# B&R Automation Studio project mappLogbook
Automation Studio 4.7.5.60 SP; technology packages: mappView 5.11.3

## Configuration PC

CPU X20CP1583, AutomationRuntime C4.72, Build 4.1.2, Safety 0.0, Vc V4.52.0

### Task classes (Cpu.sw)
```
Cyclic#8:
  Logbook <- mappLogbook.Logbook.prg
Binaries: mvLoader, TCData, udbdef, User, asfw, OpcUaMap, iomap, sysconf, arconfig, ashwd, Role, ashwac
Libraries: runtime, AsBrStr, asieccon, fileio, IecCheck, sys_lib, ArEventLog, astime
```

### Hardware
```
X20CP1583 : X20CP1583 v1.6.0.0
  Connector IF1:
    ActivateIna = 0
  Connector IF2:
    ActivateDevice = 1
  ConfigurationID = ARuser_PC
  Simulation = 1
  VolatileGlobalPvSize = 200000
  Cyclic3Tolerance = 60000000
  FileDevice1
  FileDeviceName1 = FileDevice
  FileDevicePath1 = C:\Users\hendricksf\Desktop
  ActivateOpcUa = 1
  OpcUaInformationModels_PV_Version = 1
```

## Logical view

Binary libraries used (declarations not repeated): operator, runtime, AsIecCon, AsBrStr, IecCheck, sys_lib, ArEventLog, astime, AsHttp, standard

### Package Logical/Libraries - Globale Bibliotheken

- Visualisation Logical/mappView (not shown)

### LogTypes.typ
```iecst
TYPE
	enumLogbookState :
		( (*State machine*)
		stateWait,
		stateOpen,
		stateLatest,
		stateNext,
		stateDetails1,
		stateDetails2,
		stateDetails3,
		stateDetails4,
		stateFilter,
		statePrep,
		stateError,
		stateNone
		);
	enumSeverity :
		(
		severityNotification,
		severityInformation,
		severityWarning,
		severityError
		);
	enumLogbookType :
		(
		logAccessSecurity,
		logCommisioning,
		logConnectivity,
		logFieldbus,
		logFirewall,
		logMapp,
		logMotion,
		logSafety,
		logSystem,
		logTextSystem,
		logUnitSystem,
		logUser,
		logVisualization
		);
	enumSorting :
		(
		sortingASC,
		sortingDESC
		);
	logbookCMD : 	STRUCT  (*Command structure*)
		Refresh : BOOL; (*Read all entries*)
		Update : BOOL; (*Update entries*)
		Write : BOOL; (*Write a new entry*)
		ResetError : BOOL; (*Reset error*)
	END_STRUCT;
	logbookPAR : 	STRUCT  (*Parameter structure*)
		DateNow : DATE_AND_TIME; (*Current date and time*)
		TableConfig : STRING[100]; (*Hide unused rows*)
		EntriesMax : UINT; (*Maximum number of entries, shadow of LOGBOOK_ENTRIES_MAX*)
		FilterErrorNo : UDINT; (*Filter by error number*)
		FilterErrorText : STRING[LOGBOOK_TEXT_LEN]; (*Filter by error text*)
		FilterSeverity : ARRAY[0..3]OF BOOL := [4(TRUE)]; (*Filter by severity*)
		FilterLogbook : ARRAY[0..LOGBOOK_BOOKS_MAX]OF BOOL := [14(TRUE)]; (*Filter by logbook*)
		FilterDateStart : DATE; (*Filter by date*)
		FilterDateEnd : DATE;
		Sorting : enumSorting := sortingDESC; (*Sort date asc or desc*)
		AbortOnEntriesLimit : BOOL; (*Stop looking for additional entries when limit is reached*)
		AutoUpdate : BOOL; (*Automatically update data*)
		AutoUpdateInterval : UINT := 60; (*Interval for auto update in s*)
		WriteErrorNo : UDINT; (*Error no for new entry*)
		WriteErrorText : STRING[LOGBOOK_TEXT_LEN]; (*Error text for new entry*)
		WriteSeverity : USINT := 0; (*Error severiry for new entry*)
		WriteLogbook : UINT := 0; (*Error logbook for new entry*)
	END_STRUCT;
	logbookERR : 	STRUCT  (*Error structure*)
		State : enumLogbookState; (*State where the error occured*)
	END_STRUCT;
	logbookDAT : 	STRUCT  (*Data structure*)
		Entries : logbookENTRIES;
		EntriesTotal : UINT; (*Total number of entries*)
		CntSeverity : ARRAY[0..3]OF UINT; (*Counts by severity*)
		CntLogbook : ARRAY[0..LOGBOOK_BOOKS_MAX]OF UINT; (*Counts by logbook*)
		LastUpdate : STRING[25]; (*Last refresh run*)
	END_STRUCT;
	logbookENTRIES : 	STRUCT  (*Entries structure*)
		EventID : ARRAY[1..LOGBOOK_ENTRIES_MAX]OF DINT; (*Event ID*)
		Timestamp : ARRAY[1..LOGBOOK_ENTRIES_MAX]OF STRING[25]; (*Date and time*)
		DTsec : ARRAY[1..LOGBOOK_ENTRIES_MAX]OF UDINT; (*Date and time in sec*)
		DTmsec : ARRAY[1..LOGBOOK_ENTRIES_MAX]OF UDINT; (*Additional milliseconds*)
		Severity : ARRAY[1..LOGBOOK_ENTRIES_MAX]OF USINT; (*Severity*)
		Code : ARRAY[1..LOGBOOK_ENTRIES_MAX]OF UINT; (*Code*)
		FacilityCode : ARRAY[1..LOGBOOK_ENTRIES_MAX]OF UINT; (*Facility code*)
		LogbookName : ARRAY[1..LOGBOOK_ENTRIES_MAX]OF STRING[30]; (*Logbook text*)
		ErrorNo : ARRAY[1..LOGBOOK_ENTRIES_MAX]OF DINT; (*Error number*)
		ErrorText : ARRAY[1..LOGBOOK_ENTRIES_MAX]OF STRING[LOGBOOK_TEXT_LEN]; (*Error text*)
	END_STRUCT;
	logbookMAIN : 	STRUCT  (*Main structure*)
		CMD : logbookCMD;
		PAR : logbookPAR;
		DAT : logbookDAT;
		ERR : logbookERR;
		Status : DINT;
		StatusText : STRING[80];
	END_STRUCT;
END_TYPE
```

### LogVariables.var
```iecst
VAR
	gLogbook : logbookMAIN; (*Logbook main structure*)
END_VAR
VAR CONSTANT
	LOGBOOK_EXECUTIONS : USINT := 10; (*Executions per cycle*)
	LOGBOOK_ENTRIES_MAX : UINT := 100; (*Total number of entries*)
	LOGBOOK_BOOKS_MAX : USINT := 13; (*Total number of facilities*)
	LOGBOOK_TEXT_LEN : UINT := 200; (*Error text length*)
END_VAR
```

### Program Logical/mappLogbook/Logbook (IEC)

#### Main.st - Init, cyclic, exit code
```iecst
// --------------------------------------------------------------------------------------------------------------------
// Logbook Task
// This task reads the PLC logbook and creates the data structure to display it in mappView
// --------------------------------------------------------------------------------------------------------------------
PROGRAM _INIT
	// Set time range to all on startup
	DTGetTime_0.enable := TRUE;
	DTGetTime_0();
	gLogbook.PAR.FilterDateStart := STRING_TO_DATE('D#1999-12-31');
	gLogbook.PAR.FilterDateEnd := DT_TO_DATE(DTGetTime_0.DT1);

	// Read data after reboot
	gLogbook.CMD.Refresh := TRUE;
END_PROGRAM

PROGRAM _CYCLIC
	// Abort current update run
	IF EDGENEG(gLogbook.CMD.Refresh) THEN
		IF 	state <> stateError THEN
			gLogbook.Status := ERR_OK;
			state := stateWait;
		END_IF
	END_IF
	// Run task multiple times to speed up process
	FOR executions:=1 TO LOGBOOK_EXECUTIONS DO
		// --------------------------------------------------------------------------------------------------------------------
		// Logbook state machine
		// --------------------------------------------------------------------------------------------------------------------
		CASE state OF
			// --------------------------------------------------------------------------------------------------------------------
			// Wait for new command
			// --------------------------------------------------------------------------------------------------------------------
			stateWait:
				// --------------------------------------------------------------------------------------------------------------------
				// Get current date
				DTGetTime_0.enable := TRUE;
				DTGetTime_0();
				gLogbook.PAR.DateNow := DTGetTime_0.DT1;
				gLogbook.PAR.EntriesMax := LOGBOOK_ENTRIES_MAX;

				// --------------------------------------------------------------------------------------------------------------------
				// Refresh all logbook data
				IF gLogbook.CMD.Refresh THEN
					// Erase old data, set busy state
					brsmemset(ADR(Logbook), 0, SIZEOF(Logbook));
					brsmemset(ADR(gLogbook.DAT), 0, SIZEOF(gLogbook.DAT));
					gLogbook.Status := ERR_FUB_BUSY;
					state := stateOpen;
				END_IF

				// --------------------------------------------------------------------------------------------------------------------
				// Auto update logbook data
				IF gLogbook.PAR.AutoUpdate THEN
					AutoRefresh.IN := TRUE;
					AutoRefresh.PT := gLogbook.PAR.AutoUpdateInterval*100;
					AutoRefresh();
					IF AutoRefresh.Q THEN
						AutoRefresh(IN:= FALSE);
						gLogbook.CMD.Update := TRUE;
						state := stateNext;
					END_IF
				ELSE
					AutoRefresh(IN:= FALSE);
				END_IF

				// --------------------------------------------------------------------------------------------------------------------
				// Update only latest logbook data
				IF gLogbook.CMD.Update THEN
					brsmemset(ADR(Logbook.RecordIDIsLast), 0, SIZEOF(Logbook.RecordIDIsLast));
					brsmemset(ADR(Logbook.RecordID), 0, SIZEOF(Logbook.RecordID));
					// Start at the beginning set busy state
					Logbook.CntLogbook := 0;
					gLogbook.Status := ERR_FUB_BUSY;
					state := stateLatest;
				END_IF

				// --------------------------------------------------------------------------------------------------------------------
				// Reset function blocks
				ArEventLogGetIdent_0(Execute := FALSE);
				ArEventLogGetLatestRecordID_0(Execute := FALSE);
				ArEventLogGetPreviousRecordID_0(Execute := FALSE);
				ArEventLogRead_0(Execute := FALSE);
				ArEventLogReadErrorNumber_0(Execute := FALSE);
				ArEventLogReadDescription_0(Execute := FALSE);
				ArEventLogReadAddData_0(Execute := FALSE);

				// --------------------------------------------------------------------------------------------------------------------
				// Show status, reset error command
				gLogbook.CMD.ResetError := FALSE;
				gLogbook.StatusText := 'Waiting...last update ';
				brsstrcat(ADR(gLogbook.StatusText), ADR(gLogbook.DAT.LastUpdate));
				EXIT;
				// --------------------------------------------------------------------------------------------------------------------
				// Open logbook
				// --------------------------------------------------------------------------------------------------------------------
			stateOpen:
				// Last logbook reached
				IF Logbook.CntLogbook > LOGBOOK_BOOKS_MAX THEN
					Logbook.CntLogbook := 0;
					state := stateLatest;
					EXIT;
				END_IF
				ArEventLogGetIdent_0.Execute := gLogbook.CMD.Refresh;
				ArEventLogGetIdent_0.Name := LOGBOOK_NAMES[Logbook.CntLogbook];
				ArEventLogGetIdent_0();

				// Success
				IF (ArEventLogGetIdent_0.Done AND ArEventLogGetIdent_0.StatusID = ERR_OK) OR ArEventLogGetIdent_0.StatusID = arEVENTLOG_ERR_LOGBOOK_NOT_FOUND THEN
					Logbook.Ident[Logbook.CntLogbook] := ArEventLogGetIdent_0.Ident;
					Logbook.CntLogbook := Logbook.CntLogbook + 1;
					ArEventLogGetIdent_0(Execute := FALSE);
					// Error
				ELSIF ArEventLogGetIdent_0.Error THEN
					gLogbook.ERR.State := state;
					gLogbook.Status := ArEventLogGetIdent_0.StatusID;
					state := stateError;
				END_IF
				// --------------------------------------------------------------------------------------------------------------------
				// Read latest entry
				// --------------------------------------------------------------------------------------------------------------------
			stateLatest:
				ArEventLogGetLatestRecordID_0.Execute := TRUE;
				ArEventLogGetLatestRecordID_0.Ident := Logbook.Ident[Logbook.CntLogbook];
				ArEventLogGetLatestRecordID_0();

				// Success
				IF ArEventLogGetLatestRecordID_0.Done AND ArEventLogGetLatestRecordID_0.StatusID = ERR_OK THEN
					// Store this record ID for next step
					Logbook.RecordID[Logbook.CntLogbook] := ArEventLogGetLatestRecordID_0.RecordID;
					// If there is a new entry
					IF ArEventLogGetLatestRecordID_0.RecordID > Logbook.RecordIDOld[Logbook.CntLogbook] THEN
						// Store latest ID for next update command, reset is last flag
						Logbook.RecordIDLatest[Logbook.CntLogbook] := ArEventLogGetLatestRecordID_0.RecordID;
						state := stateDetails1;
						// No new entry
					ELSE
						Logbook.RecordIDIsLast[Logbook.CntLogbook] := TRUE;
						state := statePrep;
					END_IF
					// Error
				ELSIF ArEventLogGetLatestRecordID_0.Error THEN
					gLogbook.ERR.State := state;
					gLogbook.Status := ArEventLogGetLatestRecordID_0.StatusID;
					state := stateError;
				END_IF
				// --------------------------------------------------------------------------------------------------------------------
				// Read next entry
				// --------------------------------------------------------------------------------------------------------------------
			stateNext:
				animation := WorkingStatus(ADR(gLogbook.StatusText), ADR('reading entries...'), animation);
				ArEventLogGetPreviousRecordID_0.Execute := TRUE;
				ArEventLogGetPreviousRecordID_0.Ident := Logbook.Ident[Logbook.CntLogbook];
				ArEventLogGetPreviousRecordID_0.RecordID := Logbook.RecordID[Logbook.CntLogbook];
				ArEventLogGetPreviousRecordID_0();

				// Success
				IF ArEventLogGetPreviousRecordID_0.Done AND ArEventLogGetPreviousRecordID_0.StatusID = ERR_OK THEN
					// Store this record ID for next step
					Logbook.RecordID[Logbook.CntLogbook] := ArEventLogGetPreviousRecordID_0.PrevRecordID;
					// Stop update when previous record ID is reached
					IF Logbook.RecordID[Logbook.CntLogbook] = Logbook.RecordIDOld[Logbook.CntLogbook] AND gLogbook.CMD.Update THEN
						// Remember latest entry, set is last flag
						Logbook.RecordIDOld[Logbook.CntLogbook] := Logbook.RecordIDLatest[Logbook.CntLogbook];
						Logbook.RecordIDIsLast[Logbook.CntLogbook] := TRUE;
						state := statePrep;
					ELSE
						state := stateDetails1;
					END_IF
					// Error
				ELSIF ArEventLogGetPreviousRecordID_0.Error THEN
					// Last entry reached is not an error
					IF ArEventLogGetPreviousRecordID_0.StatusID = arEVENTLOG_ERR_RECORDID_INVALID THEN
						// Remember latest entry, set is last flag
						Logbook.RecordIDOld[Logbook.CntLogbook] := Logbook.RecordIDLatest[Logbook.CntLogbook];
						Logbook.RecordIDIsLast[Logbook.CntLogbook] := TRUE;
						state := statePrep;
						// Everything else is an error
					ELSE
						gLogbook.ERR.State := state;
						gLogbook.Status := ArEventLogGetPreviousRecordID_0.StatusID;
						state := stateError;
					END_IF
				END_IF
				// --------------------------------------------------------------------------------------------------------------------
				// Read event id and time stamp
				// --------------------------------------------------------------------------------------------------------------------
			stateDetails1:
				ArEventLogRead_0.Execute := TRUE;
				ArEventLogRead_0.Ident := Logbook.Ident[Logbook.CntLogbook];
				ArEventLogRead_0.RecordID := Logbook.RecordID[Logbook.CntLogbook];
				ArEventLogRead_0();

				// Success
				IF ArEventLogRead_0.Done AND (ArEventLogRead_0.StatusID = ERR_OK OR ArEventLogRead_0.StatusID = arEVENTLOG_WRN_NO_EVENTID) THEN
					state := stateDetails2;
					// Error
				ELSIF ArEventLogRead_0.Error THEN
					gLogbook.ERR.State := state;
					gLogbook.Status := ArEventLogRead_0.StatusID;
					state := stateError;
				END_IF
				// --------------------------------------------------------------------------------------------------------------------
				// Read error no
				// --------------------------------------------------------------------------------------------------------------------
			stateDetails2:
				ArEventLogReadErrorNumber_0.Execute := TRUE;
				ArEventLogReadErrorNumber_0.Ident := Logbook.Ident[Logbook.CntLogbook];
				ArEventLogReadErrorNumber_0.RecordID := Logbook.RecordID[Logbook.CntLogbook];
				ArEventLogReadErrorNumber_0();

				// Success
				IF (ArEventLogReadErrorNumber_0.Done AND ArEventLogReadErrorNumber_0.StatusID = ERR_OK) OR ArEventLogReadErrorNumber_0.StatusID = arEVENTLOG_ERR_NO_ERRORNUMBER THEN
					state := stateDetails3;
					// Error
				ELSIF ArEventLogReadErrorNumber_0.Error THEN
					gLogbook.ERR.State := state;
					gLogbook.Status := ArEventLogReadErrorNumber_0.StatusID;
					state := stateError;
				END_IF
				// --------------------------------------------------------------------------------------------------------------------
				// Read error description
				// --------------------------------------------------------------------------------------------------------------------
			stateDetails3:
				ArEventLogReadDescription_0.Execute := TRUE;
				ArEventLogReadDescription_0.Ident := Logbook.Ident[Logbook.CntLogbook];
				ArEventLogReadDescription_0.RecordID := Logbook.RecordID[Logbook.CntLogbook];
				ArEventLogReadDescription_0.TextBuffer := ADR(ErrorText);
				ArEventLogReadDescription_0.TextBufferSize := SIZEOF(ErrorText);
				ArEventLogReadDescription_0();

				// Success
				IF (ArEventLogReadDescription_0.Done AND (ArEventLogReadDescription_0.StatusID = ERR_OK OR ArEventLogReadDescription_0.StatusID = arEVENTLOG_WRN_NO_EVENTID)) OR ArEventLogReadDescription_0.StatusID = arEVENTLOG_ERR_NO_DESCRIPTION THEN
					state := stateDetails4;
					// Error
				ELSIF ArEventLogReadDescription_0.Error THEN
					gLogbook.ERR.State := state;
					gLogbook.Status := ArEventLogReadDescription_0.StatusID;
					state := stateError;
				END_IF
				// --------------------------------------------------------------------------------------------------------------------
				// Read additional information
				// --------------------------------------------------------------------------------------------------------------------
			stateDetails4:
				// Skip if no additional data is available
				IF ArEventLogRead_0.AddDataSize > 0 THEN
					// Read additional data
					ArEventLogReadAddData_0.Execute := TRUE;
					ArEventLogReadAddData_0.Ident := Logbook.Ident[Logbook.CntLogbook];
					ArEventLogReadAddData_0.RecordID := Logbook.RecordID[Logbook.CntLogbook];
					ArEventLogReadAddData_0.AddData := ADR(AddData);
					// Limit buffer to max size
					IF ArEventLogRead_0.AddDataSize < SIZEOF(AddData) THEN
						ArEventLogReadAddData_0.BytesToRead := ArEventLogRead_0.AddDataSize;
					ELSE
						ArEventLogReadAddData_0.BytesToRead := SIZEOF(AddData);
					END_IF
					ArEventLogReadAddData_0();

					// Success
					IF (ArEventLogReadAddData_0.Done AND ArEventLogReadAddData_0.StatusID = ERR_OK) OR ArEventLogReadAddData_0.StatusID = arEVENTLOG_INF_SIZE THEN
						// Enter standard text if additional does not fit
						IF ArEventLogReadAddData_0.StatusID = arEVENTLOG_INF_SIZE THEN
							brsstrcat(ADR(ErrorText), ADR('\n >>> '));
							brsstrcat(ADR(ErrorText), ADR('Additional buffer is too small'));
						ELSE
							// Make sure string is readable
							IF brsstrcmp(ADR(AddData), ADR('')) <> 0 AND ArEventLogRead_0.AddDataFormat = arEVENTLOG_ADDFORMAT_TEXT THEN
								brsstrcat(ADR(ErrorText), ADR('\n >>> '));
								// Limit additional text to max size
								IF ArEventLogReadAddData_0.AddDataSize < SIZEOF(ErrorText) - brsstrlen(ADR(ErrorText)) THEN
									brsstrcat(ADR(ErrorText), ADR(AddData));
								ELSE
									brsmemcpy(ADR(ErrorText) + brsstrlen(ADR(ErrorText)), ADR(AddData), SIZEOF(ErrorText) - brsstrlen(ADR(ErrorText)));
								END_IF
							END_IF
						END_IF
						state := stateFilter;
						// Error
					ELSIF ArEventLogReadDescription_0.Error THEN
						gLogbook.ERR.State := state;
						gLogbook.Status := ArEventLogReadAddData_0.StatusID;
						state := stateError;
					END_IF
				ELSE
					state := stateFilter;
				END_IF
				// --------------------------------------------------------------------------------------------------------------------
				// Apply filter settings
				// --------------------------------------------------------------------------------------------------------------------
			stateFilter:
				// --------------------------------------------------------------------------------------------------------------------
				// Filters
				cntFilterNo := 0;
				cntFilterText := 0;
				cntFilterLogbook := 0;
				cntFilterSeverity := 0;
				cntFilterDate := 0;
				// --------------------------------------------------------------------------------------------------------------------
				// Check if logbook should be read
				IF  gLogbook.PAR.FilterLogbook[Logbook.CntLogbook] THEN
					cntFilterLogbook := cntFilterLogbook + 1;
				END_IF
				// --------------------------------------------------------------------------------------------------------------------
				// Check if error text matches search string
				IF gLogbook.PAR.FilterErrorText = '' OR IsInstr(ADR(ErrorText), ADR(gLogbook.PAR.FilterErrorText)) THEN
					cntFilterText := cntFilterText + 1;
				END_IF
				// --------------------------------------------------------------------------------------------------------------------
				// Make sure error number matches filter
				IF gLogbook.PAR.FilterErrorNo = 0 OR gLogbook.PAR.FilterErrorNo = ArEventLogReadErrorNumber_0.ErrorNumber THEN
					cntFilterNo := cntFilterNo + 1;
				END_IF
				// --------------------------------------------------------------------------------------------------------------------
				// Check severity filter settings
				IF ArEventLogRead_0.EventID <> 0 THEN
					gLogbook.DAT.CntSeverity[GetSeverity(EventID := ArEventLogRead_0.EventID)] := gLogbook.DAT.CntSeverity[GetSeverity(EventID := ArEventLogRead_0.EventID)] + 1;
					IF gLogbook.PAR.FilterSeverity[GetSeverity(EventID := ArEventLogRead_0.EventID)] THEN
						cntFilterSeverity := cntFilterSeverity + 1;
					END_IF
				ELSE
					gLogbook.DAT.CntSeverity[ArEventLogReadErrorNumber_0.Severity] := gLogbook.DAT.CntSeverity[ArEventLogReadErrorNumber_0.Severity] + 1;
					IF gLogbook.PAR.FilterSeverity[ArEventLogReadErrorNumber_0.Severity] THEN
						cntFilterSeverity := cntFilterSeverity + 1;
					END_IF
				END_IF
				// --------------------------------------------------------------------------------------------------------------------
				// Check date range
				tmpSTR:= DT_TO_STRING(DATE_TO_DT(gLogbook.PAR.FilterDateStart));
				brsmemcpy(ADR(tmpSTR)+13, ADR('-00:00:00'), 9);
				TimeStart := STRING_TO_DT(tmpSTR);
				tmpSTR:= DT_TO_STRING(DATE_TO_DT(gLogbook.PAR.FilterDateEnd));
				brsmemcpy(ADR(tmpSTR)+13, ADR('-23:59:59'), 9);
				TimeEnd := STRING_TO_DT(tmpSTR);
				IF ArEventLogRead_0.TimeStamp.sec >= DT_TO_UDINT(TimeStart) AND ArEventLogRead_0.TimeStamp.sec <= DT_TO_UDINT(TimeEnd) THEN
					cntFilterDate := cntFilterDate + 1;
				END_IF
				// --------------------------------------------------------------------------------------------------------------------
				// Count logbook entries
				gLogbook.DAT.CntLogbook[Logbook.CntLogbook] := gLogbook.DAT.CntLogbook[Logbook.CntLogbook] +  1;

				// --------------------------------------------------------------------------------------------------------------------
				// Transfer data
				IF cntFilterNo > 0 AND cntFilterText > 0 AND cntFilterLogbook > 0 AND cntFilterSeverity > 0 AND cntFilterDate > 0 THEN
					// --------------------------------------------------------------------------------------------------------------------
					// Find new place for entry
					idx := InsertEntry(ADR(gLogbook.DAT), ArEventLogRead_0.TimeStamp.sec, UDINT_TO_UINT(ArEventLogRead_0.TimeStamp.nsec/1000000), gLogbook.PAR.Sorting);
					IF idx <> NO_SPACE THEN
						// Store date and time
						gLogbook.DAT.Entries.DTsec[idx] := ArEventLogRead_0.TimeStamp.sec;
						gLogbook.DAT.Entries.DTmsec[idx] := UDINT_TO_UINT(ArEventLogRead_0.TimeStamp.nsec/1000000);
						// Add timestamp
						tmpDT := UDINT_TO_DT(ArEventLogRead_0.TimeStamp.sec);
						DT_TO_DTStructure(tmpDT, ADR(tmpDTstruct));
						brsmemset(ADR(gLogbook.DAT.Entries.Timestamp[idx]), 0, SIZEOF(gLogbook.DAT.Entries.Timestamp[idx]));
						NormalizeDateTime(ADR(gLogbook.DAT.Entries.Timestamp[idx]), tmpDTstruct.day, '');
						NormalizeDateTime(ADR(gLogbook.DAT.Entries.Timestamp[idx]), tmpDTstruct.month, '.');
						NormalizeDateTime(ADR(gLogbook.DAT.Entries.Timestamp[idx]), tmpDTstruct.year, '.');
						NormalizeDateTime(ADR(gLogbook.DAT.Entries.Timestamp[idx]), tmpDTstruct.hour, ' ');
						NormalizeDateTime(ADR(gLogbook.DAT.Entries.Timestamp[idx]), tmpDTstruct.minute, ':');
						NormalizeDateTime(ADR(gLogbook.DAT.Entries.Timestamp[idx]), tmpDTstruct.second, ':');
						NormalizeDateTime(ADR(gLogbook.DAT.Entries.Timestamp[idx]), gLogbook.DAT.Entries.DTmsec[idx], '.');
						// Add event ID, code, logbook, severity
						gLogbook.DAT.Entries.EventID[gLogbook.DAT.EntriesTotal] := ArEventLogRead_0.EventID;
						IF ArEventLogRead_0.EventID <> 0 THEN
							gLogbook.DAT.Entries.Severity[idx] := GetSeverity(EventID := ArEventLogRead_0.EventID);
						ELSE
							gLogbook.DAT.Entries.Severity[idx] := ArEventLogReadErrorNumber_0.Severity;
						END_IF
						gLogbook.DAT.Entries.Code[idx] := GetCode(EventID := ArEventLogRead_0.EventID);
						gLogbook.DAT.Entries.FacilityCode[idx] := GetFacility(EventID := ArEventLogRead_0.EventID);
						gLogbook.DAT.Entries.LogbookName[idx] := LOGBOOK_TEXT[Logbook.CntLogbook];
						// Add error number and text, use event ID if error no is 0
						IF ArEventLogReadErrorNumber_0.ErrorNumber <> 0 THEN
							gLogbook.DAT.Entries.ErrorNo[idx] := ArEventLogReadErrorNumber_0.ErrorNumber;
						ELSE
							gLogbook.DAT.Entries.ErrorNo[idx] := ArEventLogRead_0.EventID;
						END_IF
						httpUtf8ToString_0(enable := TRUE, pSrc := ADR(ErrorText), pDest := ADR(gLogbook.DAT.Entries.ErrorText[idx]), destSize := SIZEOF(gLogbook.DAT.Entries.ErrorText[idx]));
					END_IF
				END_IF

				// --------------------------------------------------------------------------------------------------------------------
				// Hide unused table rows
				brsitoa(gLogbook.DAT.EntriesTotal, ADR(tmpSTR));
				gLogbook.PAR.TableConfig := '{"specRows":[{"from":';
				brsstrcat(ADR(gLogbook.PAR.TableConfig), ADR(tmpSTR));
				brsstrcat(ADR(gLogbook.PAR.TableConfig), ADR(', "to":'));
				brsitoa(LOGBOOK_ENTRIES_MAX, ADR(tmpSTR));
				brsstrcat(ADR(gLogbook.PAR.TableConfig), ADR(tmpSTR));
				brsstrcat(ADR(gLogbook.PAR.TableConfig), ADR(', "visible":false}]}'));

				state := statePrep;

				// --------------------------------------------------------------------------------------------------------------------
				// Perpare for next entry
				// --------------------------------------------------------------------------------------------------------------------
			statePrep:
				// --------------------------------------------------------------------------------------------------------------------
				// Reset buffer and function blocks
				brsmemset(ADR(AddData), 0, SIZEOF(AddData));
				ArEventLogGetLatestRecordID_0(Execute := FALSE);
				ArEventLogGetPreviousRecordID_0(Execute := FALSE);
				ArEventLogRead_0(Execute := FALSE);
				ArEventLogReadErrorNumber_0(Execute := FALSE);
				ArEventLogReadDescription_0(Execute := FALSE);
				ArEventLogReadAddData_0(Execute := FALSE);

				// --------------------------------------------------------------------------------------------------------------------
				// Find next logbook from here to the end
				REPEAT
					Logbook.CntLogbook := Logbook.CntLogbook + 1;
					IF Logbook.CntLogbook <= LOGBOOK_BOOKS_MAX THEN
						IF (Logbook.Ident[Logbook.CntLogbook] <> 0 AND NOT Logbook.RecordIDIsLast[Logbook.CntLogbook]) OR (Logbook.Ident[Logbook.CntLogbook] <> 0 AND Logbook.RecordID[Logbook.CntLogbook] = 0) THEN
							EXIT;
						END_IF
					END_IF
					UNTIL Logbook.CntLogbook > LOGBOOK_BOOKS_MAX
				END_REPEAT;

				// --------------------------------------------------------------------------------------------------------------------
				// No logbook found, start at the beginning
				IF Logbook.CntLogbook > LOGBOOK_BOOKS_MAX THEN
					Logbook.CntLogbook := 0;
					// Find next logbook from start to the end
					REPEAT
						IF (Logbook.Ident[Logbook.CntLogbook] <> 0 AND NOT Logbook.RecordIDIsLast[Logbook.CntLogbook]) OR (Logbook.Ident[Logbook.CntLogbook] <> 0 AND Logbook.RecordID[Logbook.CntLogbook] = 0) THEN
							EXIT;
						END_IF
						Logbook.CntLogbook := Logbook.CntLogbook + 1;
						UNTIL Logbook.CntLogbook > LOGBOOK_BOOKS_MAX
					END_REPEAT;
				END_IF

				// --------------------------------------------------------------------------------------------------------------------
				// Finish when no logbook found or max entries is reached
				IF Logbook.CntLogbook > LOGBOOK_BOOKS_MAX OR (gLogbook.PAR.AbortOnEntriesLimit AND gLogbook.DAT.EntriesTotal = LOGBOOK_ENTRIES_MAX) THEN
					// Add last update
					DT_TO_DTStructure(gLogbook.PAR.DateNow, ADR(tmpDTstruct));
					brsmemset(ADR(gLogbook.DAT.LastUpdate), 0, SIZEOF(gLogbook.DAT.LastUpdate));
					NormalizeDateTime(ADR(gLogbook.DAT.LastUpdate), tmpDTstruct.day, '');
					NormalizeDateTime(ADR(gLogbook.DAT.LastUpdate), tmpDTstruct.month, '.');
					NormalizeDateTime(ADR(gLogbook.DAT.LastUpdate), tmpDTstruct.year, '.');
					NormalizeDateTime(ADR(gLogbook.DAT.LastUpdate), tmpDTstruct.hour, ' ');
					NormalizeDateTime(ADR(gLogbook.DAT.LastUpdate), tmpDTstruct.minute, ':');
					NormalizeDateTime(ADR(gLogbook.DAT.LastUpdate), tmpDTstruct.second, ':');
					// Reset status and command
					gLogbook.Status := ERR_OK;
					gLogbook.CMD.Refresh := FALSE;
					gLogbook.CMD.Update := FALSE;
					state := stateWait;
				ELSE
					// Read latest entry
					IF Logbook.RecordID[Logbook.CntLogbook] = 0 THEN
						state := stateLatest;
						// Read next entry
					ELSE
						state := stateNext;
					END_IF
				END_IF

				// --------------------------------------------------------------------------------------------------------------------
				// Error state
				// --------------------------------------------------------------------------------------------------------------------
			stateError:
				gLogbook.StatusText := 'Error...';
				brsmemset(ADR(gLogbook.CMD), 0, SIZEOF(gLogbook.CMD)-1);
				// Reset error
				IF gLogbook.CMD.ResetError THEN
					gLogbook.ERR.State := stateNone;
					gLogbook.Status := 0;
					gLogbook.CMD.ResetError := FALSE;
					state := stateWait;
				END_IF
				EXIT;
		END_CASE;
	END_FOR;

END_PROGRAM
```

#### Variables.var - Local variables
```iecst
(*---------------------------------------------------------------------------------------------------------------------------------*)
VAR
	ErrorText : STRING[LOGBOOK_TEXT_LEN];
	cntFilterNo : UINT;
	cntFilterText : UINT;
	cntFilterLogbook : UINT;
	cntFilterSeverity : UINT;
	cntFilterDate : UINT;
	tmpSTR : STRING[100];
	tmpDT : DATE_AND_TIME;
	tmpDTstruct : DTStructure;
	TimeStart : DATE_AND_TIME;
	TimeEnd : DATE_AND_TIME;
	AddData : ARRAY[0..500] OF USINT;
	Logbook : typLogbook;
	idx : UINT;
	animation : USINT;
END_VAR
(*---------------------------------------------------------------------------------------------------------------------------------*)
(*Local function*)
VAR
	ArEventLogGetPreviousRecordID_0 : ArEventLogGetPreviousRecordID;
	ArEventLogGetLatestRecordID_0 : ArEventLogGetLatestRecordID;
	ArEventLogRead_0 : ArEventLogRead;
	ArEventLogReadErrorNumber_0 : ArEventLogReadErrorNumber;
	ArEventLogReadDescription_0 : ArEventLogReadDescription;
	ArEventLogReadAddData_0 : ArEventLogReadAddData;
	DTGetTime_0 : DTGetTime;
	httpUtf8ToString_0 : httpUtf8ToString;
	AutoRefresh : TON_10ms;
END_VAR
(*Local variables*)
VAR
	state : enumLogbookState;
	ArEventLogGetIdent_0 : ArEventLogGetIdent;
	executions : USINT;
END_VAR
(*---------------------------------------------------------------------------------------------------------------------------------*)
(*Local constants*)
VAR CONSTANT
	LOGBOOK_NAMES : ARRAY[0..LOGBOOK_BOOKS_MAX] OF STRING[50] := ['$$accsec','$$diag','$$arlogconn','$$fieldbus','$$firewall','$$mapp','$$motion','$$safety','$$arlogsys','$$textsys','$$unitsys','$$arlogusr','$$vision','$$visu'];
	LOGBOOK_TEXT : ARRAY[0..LOGBOOK_BOOKS_MAX] OF STRING[50] := ['Access','Commissioning','Connectivity','Fieldbus','Firewall','Mapp','Motion','Safety','System','Text System','Unit System','User','Vision','Visualization'];
	NO_SPACE : UINT := 0;
END_VAR
```

#### Types.typ
```iecst
TYPE
	typLogbook : 	STRUCT
		Ident : ARRAY[0..LOGBOOK_BOOKS_MAX]OF UDINT;
		RecordIDLatest : ARRAY[0..LOGBOOK_BOOKS_MAX]OF UDINT;
		RecordIDOld : ARRAY[0..LOGBOOK_BOOKS_MAX]OF UDINT;
		RecordIDIsLast : ARRAY[0..LOGBOOK_BOOKS_MAX]OF BOOL;
		RecordID : ARRAY[0..LOGBOOK_BOOKS_MAX]OF UDINT;
		CntLogbook : USINT;
	END_STRUCT;
END_TYPE
```

#### LocalFunctions.fun
```iecst
FUNCTION GetSeverity : USINT
	VAR_INPUT
		EventID : DINT;
	END_VAR
END_FUNCTION

FUNCTION GetFacility : UINT
	VAR_INPUT
		EventID : DINT;
	END_VAR
END_FUNCTION

{REDUND_ERROR} FUNCTION GetCode : UINT (*create mappView string data provider*) (*$GROUP=User,$CAT=User,$GROUPICON=User.png,$CATICON=User.png*)
	VAR_INPUT
		EventID : DINT;
	END_VAR
END_FUNCTION

FUNCTION InsertEntry : UINT
	VAR_INPUT
		DAT : REFERENCE TO logbookDAT;
		DTsec : UDINT;
		DTmsec : UINT;
		Sorting : enumSorting;
	END_VAR
	VAR
		idx : UINT;
		idy : UINT;
	END_VAR
END_FUNCTION

FUNCTION NormalizeDateTime : UDINT
	VAR_INPUT
		target : UDINT;
		value : UDINT;
		addSTR : STRING[5];
	END_VAR
	VAR
		tmpSTR1 : STRING[10];
		tmpSTR2 : STRING[10];
	END_VAR
END_FUNCTION

FUNCTION WorkingStatus : USINT
	VAR_INPUT
		target : UDINT;
		text : UDINT;
		animation : USINT;
	END_VAR
END_FUNCTION

FUNCTION IsInstr : BOOL
	VAR_INPUT
		string1 : UDINT;
		string2 : UDINT;
	END_VAR
	VAR
		idx : UDINT;
	END_VAR
END_FUNCTION
```

#### LocalFunctions.st
```iecst
// --------------------------------------------------------------------------------------------------------------------
// Gets severity from EventId (bits 31-30)
FUNCTION GetSeverity
	IF ArEventLogIsError(EventID := EventID) THEN
		GetSeverity := arEVENTLOG_SEVERITY_ERROR;
	ELSIF ArEventLogIsWarning(EventID := EventID) THEN
		GetSeverity := arEVENTLOG_SEVERITY_WARNING;
	ELSIF ArEventLogIsInformation(EventID := EventID) THEN
		GetSeverity := arEVENTLOG_SEVERITY_INFO;
	ELSIF ArEventLogIsSuccess(EventID := EventID) THEN
		GetSeverity := arEVENTLOG_SEVERITY_SUCCESS;
	END_IF
END_FUNCTION

// --------------------------------------------------------------------------------------------------------------------
// Gets code from EventId (bits 15-0)
FUNCTION GetCode
	GetCode := DINT_TO_UINT(EventID);
END_FUNCTION

// --------------------------------------------------------------------------------------------------------------------
// Gets facility from EventId (bits 27-16)
FUNCTION GetFacility
	GetFacility := DINT_TO_UINT(SHR(EventID, 16) AND 16#0FFF);
END_FUNCTION

// --------------------------------------------------------------------------------------------------------------------
// --------------------------------------------------------------------------------------------------------------------
// Insert new entry
FUNCTION InsertEntry
	// Lets see where new entry fits
	FOR idx:=1 TO DAT.EntriesTotal DO
		// Sorting is ascending
		IF Sorting = sortingASC THEN
			// New entry is old than this entry
			IF DTsec < DAT.Entries.DTsec[idx] THEN
				EXIT;
				// If entries are within the same second check milisecond data
			ELSIF DTsec = DAT.Entries.DTsec[idx] THEN
				IF DTmsec < DAT.Entries.DTmsec[idx] THEN
					EXIT;
				END_IF
			END_IF
			// Sorting is descending
		ELSE
			// New entry is newer than this entry
			IF DTsec > DAT.Entries.DTsec[idx] THEN
				EXIT;
				// If entries are within the same second check milisecond data
			ELSIF DTsec = DAT.Entries.DTsec[idx] THEN
				IF DTmsec > DAT.Entries.DTmsec[idx] THEN
					EXIT;
				END_IF
			END_IF
		END_IF
	END_FOR;

	// Add data as long as buffer is not full
	IF DAT.EntriesTotal < LOGBOOK_ENTRIES_MAX THEN
		IF DAT.EntriesTotal = 1 AND idx = 1 THEN
			idy := 1;
		ELSIF DAT.EntriesTotal > idx THEN
			idy := DAT.EntriesTotal - idx + 1;
		END_IF
		DAT.EntriesTotal := DAT.EntriesTotal + 1;
		// If buffer is full check where entry fits
	ELSE
		// Entry is beyond scope of buffer
		IF idx > LOGBOOK_ENTRIES_MAX THEN
			InsertEntry := NO_SPACE;
			RETURN;
		ELSE
			IF DAT.EntriesTotal - idx > 0 THEN
				idy := DAT.EntriesTotal - idx;
			END_IF
		END_IF
	END_IF

	// Dont move if there is nothing to move
	IF idy <> 0 THEN
		brsmemmove(ADR(DAT.Entries.Code[idx+1]),ADR(DAT.Entries.Code[idx]), idy * SIZEOF(DAT.Entries.Code[1]));
		brsmemmove(ADR(DAT.Entries.Timestamp[idx+1]),ADR(DAT.Entries.Timestamp[idx]), idy * SIZEOF(DAT.Entries.Timestamp[1]));
		brsmemmove(ADR(DAT.Entries.DTsec[idx+1]),ADR(DAT.Entries.DTsec[idx]), idy * SIZEOF(DAT.Entries.DTsec[1]));
		brsmemmove(ADR(DAT.Entries.DTmsec[idx+1]),ADR(DAT.Entries.DTmsec[idx]), idy * SIZEOF(DAT.Entries.DTmsec[1]));
		brsmemmove(ADR(DAT.Entries.ErrorNo[idx+1]),ADR(DAT.Entries.ErrorNo[idx]), idy * SIZEOF(DAT.Entries.ErrorNo[1]));
		brsmemmove(ADR(DAT.Entries.ErrorText[idx+1]),ADR(DAT.Entries.ErrorText[idx]), idy * SIZEOF(DAT.Entries.ErrorText[1]));
		brsmemmove(ADR(DAT.Entries.EventID[idx+1]),ADR(DAT.Entries.EventID[idx]), idy * SIZEOF(DAT.Entries.EventID[1]));
		brsmemmove(ADR(DAT.Entries.FacilityCode[idx+1]),ADR(DAT.Entries.FacilityCode[idx]), idy * SIZEOF(DAT.Entries.FacilityCode[1]));
		brsmemmove(ADR(DAT.Entries.LogbookName[idx+1]),ADR(DAT.Entries.LogbookName[idx]), idy * SIZEOF(DAT.Entries.LogbookName[1]));
		brsmemmove(ADR(DAT.Entries.Severity[idx+1]),ADR(DAT.Entries.Severity[idx]), idy * SIZEOF(DAT.Entries.Severity[1]));
	END_IF
	InsertEntry := idx;

END_FUNCTION

// --------------------------------------------------------------------------------------------------------------------
// Normalize 2 digit date and time values
FUNCTION NormalizeDateTime
	tmpSTR2 := addSTR;
	IF(value < 10) THEN
		brsstrcat(ADR(tmpSTR2), ADR('0'));
	END_IF
	brsitoa(value, ADR(tmpSTR1));
	brsstrcat(ADR(tmpSTR2), ADR(tmpSTR1));
	brsstrcat(target, ADR(tmpSTR2));
	NormalizeDateTime := TRUE;
END_FUNCTION

// --------------------------------------------------------------------------------------------------------------------
// Working status
FUNCTION WorkingStatus
	animation := animation+1;

	IF (animation = 80) THEN
		animation := 0;
	END_IF

	brsstrcpy(target, text);
	CASE(animation) OF
		0..19	: brsstrcat(target, ADR('/'));
		20..39	: brsstrcat(target, ADR('-'));
		40..59	: brsstrcat(target, ADR('\'));
		60..79	: brsstrcat(target, ADR('|'));
	END_CASE;
	WorkingStatus := animation;
END_FUNCTION

// --------------------------------------------------------------------------------------------------------------------
// Is second string in first string
FUNCTION IsInstr
	IF (brsstrlen(string1) > brsstrlen(string2)) THEN
		FOR idx:=0 TO brsstrlen(string1) - brsstrlen(string2) DO
			IF (brsmemcmp(string1 + idx, string2, brsstrlen(string2)) = 0) THEN
				IsInstr := TRUE;
				EXIT;
			END_IF
		END_FOR;
	END_IF
END_FUNCTION
```

### changelog.txt
```
Next Version
- Fixed desc sorting

Version 0.3
- New update table command
- New create entry command
- Add max entries to parameter structure
- Show table during run
- Renamed facility to logbook and logbook name

Version 0.2
- Fixed special characters not showing up correct
- Fixed filter checkboxes dont remember state
- Fixed last entry is not always record ID 1
- Option to stop searching when entry limit is reached
- Option to abort current update run
- Smaller bug fixes

Version 0.1
- First public release
```

Listed in the project but not available here: Logical/Global.typ, Logical/Global.var
